(* PLC project  *)

CONFIGURATION Empty_Module_13
END_CONFIGURATION
